// TIA Portal V17 export
// export: Created 2023-02-14T02:49:22.5517164Z, ExportSetting WithDefaults, DisplayName Totally Integrated Automation Portal, DisplayVersion V17, DisplayName TIA Portal Openness, DisplayVersion V17, DisplayName TIA Portal Teamcenter Gateway, DisplayVersion V17, DisplayName TIA Portal Version Control Interface, DisplayVersion V17, DisplayName SINAMICS Startdrive Advanced, DisplayVersion V17, DisplayName SINAMICS Startdrive G130, G150, S120, S150, SINAMICS MV, S210, DisplayVersion V17, DisplayName SINAMICS Startdrive G110M, G120, G120C, G120D, G120P, G115D, DisplayVersion V17, DisplayName STEP 7 Professional, DisplayVersion V17, DisplayName STEP 7 Safety, DisplayVersion V17, DisplayName WinCC Professional, DisplayVersion V17
DATA_BLOCK "Danfos_VSD_DB"   // DB46
VERSION : 0.1
// stored: AutoNumber false, DBAccessibleFromOPCUA true, DBAccessibleFromWebserver true, InstanceOfName Danfos_VSD, InstanceOfType FB
"Danfos_VSD"
   // VAR_INPUT
   //    In_CMD : Bool;
   //    Reset : Bool;
   //    QuickStop : Bool;
   //    drive_f_setpoint : Real;
   //    In_STW : Word;
   //    drive_AV { ExternalAccessible := 'False'; ExternalVisible := 'False'; ExternalWritable := 'False'} : Int;
   // END_VAR
   // VAR_OUTPUT
   //    Danfos_CTW : Word;
   //    Danfos_SP { ExternalAccessible := 'False'; ExternalVisible := 'False'; ExternalWritable := 'False'} : Word;
   //    Drive_OK : Bool;
   //    Drive_Run : Bool;
   //    QAlarm : Word;
   //    Danfos_f_act : Real;
   //    "Danfos_QAV_%" : Real;
   // END_VAR
   // VAR
   //    SW : Struct
   //       "Bit 0-Control" : Bool;
   //       "Bit 1-Drive" : Bool;
   //       "Bit 2-Coasting stop" : Bool;
   //       "Bit 3-Trip" : Bool;
   //       "Bit 4-Error" : Bool;
   //       "Bit 5-NOP" : Bool;
   //       "Bit 6-triplock" : Bool;
   //       "Bit 7-Warning" : Bool;
   //       "Bit 8-Speed reference" : Bool;
   //       "Bit 9-Operation" : Bool;
   //       "Bit 10-frequency range" : Bool;
   //       "Bit 11-Operation" : Bool;
   //       "Bit 12-Drive OK" : Bool;
   //       "Bit 13-Voltage OK" : Bool;
   //       "Bit 14-Torque OK" : Bool;
   //       "Bit 15-Timers OK" : Bool;
   //    END_STRUCT;
   //    Reset_PE : Bool;
   //    Reset_Bits : Bool;
   //    f_act : Real;
   // END_VAR
BEGIN
END_DATA_BLOCK
